// TIA Portal V18 program export: 3 tag tables, 0 data types, 3 data blocks, 3 code blocks (in call order from the OBs), 0 instance data blocks

VAR_GLOBAL   // PLC tag table "Default tag table"
   Motor_Contactor AT %Q0.0 : Bool;
   Clock_Byte AT %MB100 : Byte;
   Clock_10Hz AT %M100.0 : Bool;
   Clock_5Hz AT %M100.1 : Bool;
   "Clock_2.5Hz" AT %M100.2 : Bool;
   Clock_2Hz AT %M100.3 : Bool;
   "Clock_1.25Hz" AT %M100.4 : Bool;
   "Clock_0.625Hz" AT %M100.6 : Bool;
   "Clock_0.5Hz" AT %M100.7 : Bool;
END_VAR

VAR_GLOBAL   // PLC tag table "Encoder_Tags"
   HSC_1_Value AT %ID1000 : DInt;   // Giá trị đếm xung thời kỳ thực từ bộ đếm tốc độ cao HSC1   {ExternalWritable false}
END_VAR

VAR_GLOBAL   // PLC tag table "PLC2_Tags"
   MB_ControlWord AT %MW40 : Word;
   MB_FreqSetpoint AT %MW42 : Int;
   MB_StatusWord AT %MW44 : Word;
   MB_ActualSpeed AT %MW46 : Int;
   MB_Error AT %M50.0 : Bool;
   MB_Busy AT %M50.1 : Bool;
   MB_Done AT %M50.2 : Bool;
   MB_Status AT %MW52 : Word;
   iStep AT %MW60 : Int;
   Freq_Temp AT %MD70 : Real;
   Speed_Actual_Temp AT %MD74 : Real;
   FirstScan AT %M101.0 : Bool;
   Clock_1Hz AT %M100.5 : Bool;
   MBCL_Done AT %M51.0 : Bool;
   MBCL_Error AT %M51.1 : Bool;
   MBCL_Status AT %MW54 : Word;
END_VAR

DATA_BLOCK "DB1_NhanTuPLC1"   // DB1
{ S7_Optimized_Access := 'FALSE' }
VERSION : 0.1
// stored: AutoNumber true, IsOnlyStoredInLoadMemory false, IsWriteProtectedInAS false
   VAR
      Speed_SP_fromPLC1 : Real;
      Control_Byte : Bool;
      Reset_Cmd : Bool;
      DIR_Cmd : Bool;
   END_VAR
BEGIN
END_DATA_BLOCK

DATA_BLOCK "DB2_GuiVePLC1"   // DB2
{ S7_Optimized_Access := 'FALSE' }
VERSION : 0.1
// stored: AutoNumber true, IsOnlyStoredInLoadMemory false, IsWriteProtectedInAS false
   VAR
      Speed_Actual_toSend : Real;
      ATV12_Status_toSend : Word;
   END_VAR
BEGIN
END_DATA_BLOCK

DATA_BLOCK "DB3_Encoder"   // DB5
TITLE = Encoder HSC Data Block
{ S7_Optimized_Access := 'FALSE' }
VERSION : 0.1
// Khối dữ liệu chứa tham số và trạng thái Encoder HSC1
// stored: AutoNumber true, IsOnlyStoredInLoadMemory false, IsWriteProtectedInAS false
   VAR
      Encoder_Count_Current : DInt;
      Encoder_Count_Last : DInt;
      Encoder_Count_Delta : DInt;
      Encoder_Count_Delta_Real : Real;
      Encoder_PPR : Real := 1000.0;
      Encoder_Effective_PPR : Real;
      Encoder_SampleTime_s : Real := 0.1;
      Encoder_RPM : Real;
      Encoder_Hz_Raw : Real;
      Encoder_Hz : Real;
      Encoder_Feedback_Selected : Real;
      Encoder_Use_Feedback : Bool := true;
      Encoder_Fault : Bool;
      Encoder_Use_Fourfold : Bool := true;
      Encoder_Motor_Pole_Pairs : Real := 2.0;
      Encoder_Fallback_Active : Bool;
      Encoder_NoPulse_Count : Real;
      Encoder_NoPulse_Limit : Real := 30.0;
   END_VAR
BEGIN
END_DATA_BLOCK

ORGANIZATION_BLOCK "Main"   // OB1, LAD, ProgramCycle
TITLE = "Main Program Sweep (Cycle)"
{ S7_Optimized_Access := 'TRUE' }
VERSION : 0.1
// stored: AutoNumber true, IsIECCheckEnabled false, SetENOAutomatically false
   VAR_INPUT
      Initial_Call : Bool;   // Initial call of this OB
      Remanence : Bool;   // =True, if remanent data are available
   END_VAR
BEGIN

REGION Network 1: Call FC_PLC2_Logic (Convert + Step Advance)
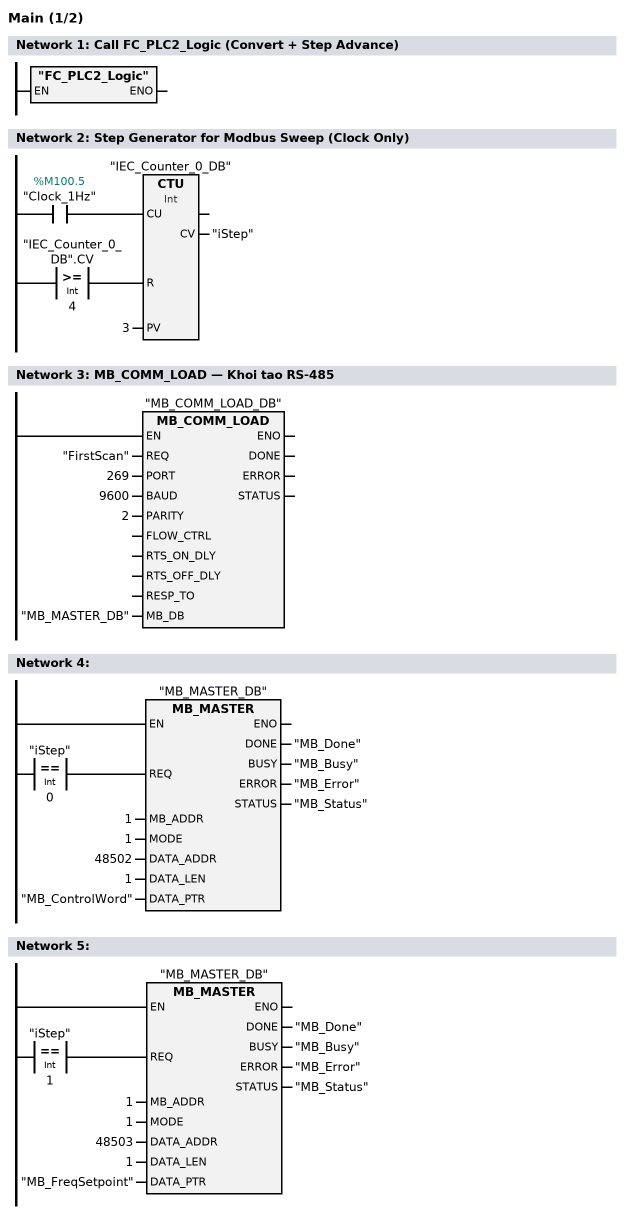
   RUNG wire#powerrail
      "FC_PLC2_Logic"()
   END_RUNG
   // the same network as SCL:
   "FC_PLC2_Logic"();
END_REGION

REGION Network 2: Step Generator for Modbus Sweep (Clock Only)
   RUNG wire#powerrail
      Contact( "Clock_1Hz" )
      { S7_Templates := "value_type := Int" } "IEC_Counter_0_DB".CTU(r := wire#w1, pv := 3, cv => "iStep")
   END_RUNG
   RUNG wire#powerrail
      { S7_Templates := "SrcType := Int" } GE_Contact(in1 := "IEC_Counter_0_DB".CV, in2 := 4)
   END_RUNG wire#w1
   // the same network as SCL:
   "IEC_Counter_0_DB".CTU(CU := "Clock_1Hz", R := "IEC_Counter_0_DB".CV >= 4, PV := 3, CV => "iStep");
END_REGION

REGION Network 3: MB_COMM_LOAD — Khoi tao RS-485
   RUNG wire#powerrail
      "MB_COMM_LOAD_DB".MB_COMM_LOAD(REQ := "FirstScan", PORT := 269, BAUD := 9600, PARITY := 2, FLOW_CTRL :=, RTS_ON_DLY :=, RTS_OFF_DLY :=, RESP_TO :=, MB_DB := "MB_MASTER_DB", DONE =>, ERROR =>, STATUS =>)
   END_RUNG
   // the same network as SCL:
   "MB_COMM_LOAD_DB"(REQ := "FirstScan", PORT := 269, BAUD := 9600, PARITY := 2, MB_DB := "MB_MASTER_DB");   // MB_COMM_LOAD
END_REGION

REGION Network 4
   RUNG wire#powerrail
      "MB_MASTER_DB".MB_MASTER(REQ := wire#w1, MB_ADDR := 1, MODE := 1, DATA_ADDR := 48502, DATA_LEN := 1, DATA_PTR := "MB_ControlWord", DONE => "MB_Done", BUSY => "MB_Busy", ERROR => "MB_Error", STATUS => "MB_Status")
   END_RUNG
   RUNG wire#powerrail
      { S7_Templates := "SrcType := Int" } EQ_Contact(in1 := "iStep", in2 := 0)
   END_RUNG wire#w1
   // the same network as SCL:
   "MB_MASTER_DB"(REQ := "iStep" = 0,   // MB_MASTER
                  MB_ADDR := 1,
                  MODE := 1,
                  DATA_ADDR := 48502,
                  DATA_LEN := 1,
                  DATA_PTR := "MB_ControlWord",
                  DONE => "MB_Done",
                  BUSY => "MB_Busy",
                  ERROR => "MB_Error",
                  STATUS => "MB_Status");
END_REGION

REGION Network 5
   RUNG wire#powerrail
      "MB_MASTER_DB".MB_MASTER(REQ := wire#w1, MB_ADDR := 1, MODE := 1, DATA_ADDR := 48503, DATA_LEN := 1, DATA_PTR := "MB_FreqSetpoint", DONE => "MB_Done", BUSY => "MB_Busy", ERROR => "MB_Error", STATUS => "MB_Status")
   END_RUNG
   RUNG wire#powerrail
      { S7_Templates := "SrcType := Int" } EQ_Contact(in1 := "iStep", in2 := 1)
   END_RUNG wire#w1
   // the same network as SCL:
   "MB_MASTER_DB"(REQ := "iStep" = 1,   // MB_MASTER
                  MB_ADDR := 1,
                  MODE := 1,
                  DATA_ADDR := 48503,
                  DATA_LEN := 1,
                  DATA_PTR := "MB_FreqSetpoint",
                  DONE => "MB_Done",
                  BUSY => "MB_Busy",
                  ERROR => "MB_Error",
                  STATUS => "MB_Status");
END_REGION

REGION Network 6
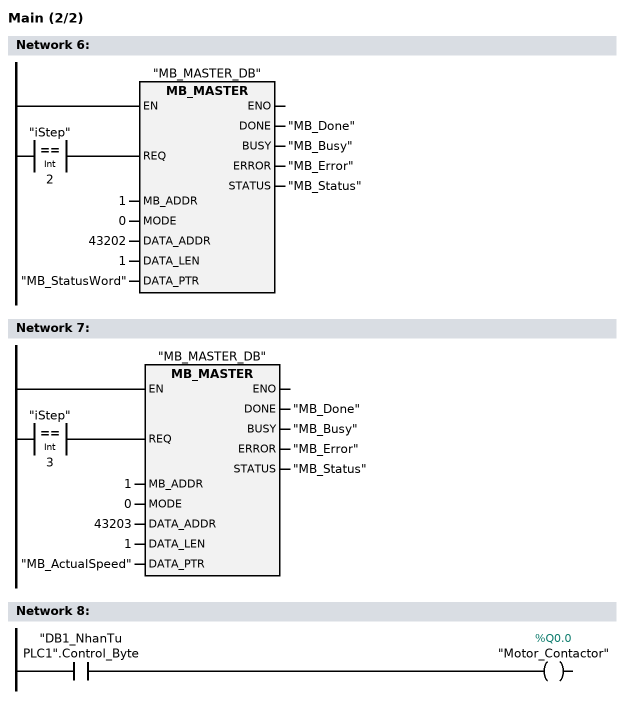
   RUNG wire#powerrail
      "MB_MASTER_DB".MB_MASTER(REQ := wire#w1, MB_ADDR := 1, MODE := 0, DATA_ADDR := 43202, DATA_LEN := 1, DATA_PTR := "MB_StatusWord", DONE => "MB_Done", BUSY => "MB_Busy", ERROR => "MB_Error", STATUS => "MB_Status")
   END_RUNG
   RUNG wire#powerrail
      { S7_Templates := "SrcType := Int" } EQ_Contact(in1 := "iStep", in2 := 2)
   END_RUNG wire#w1
   // the same network as SCL:
   "MB_MASTER_DB"(REQ := "iStep" = 2,   // MB_MASTER
                  MB_ADDR := 1,
                  MODE := 0,
                  DATA_ADDR := 43202,
                  DATA_LEN := 1,
                  DATA_PTR := "MB_StatusWord",
                  DONE => "MB_Done",
                  BUSY => "MB_Busy",
                  ERROR => "MB_Error",
                  STATUS => "MB_Status");
END_REGION

REGION Network 7
   RUNG wire#powerrail
      "MB_MASTER_DB".MB_MASTER(REQ := wire#w1, MB_ADDR := 1, MODE := 0, DATA_ADDR := 43203, DATA_LEN := 1, DATA_PTR := "MB_ActualSpeed", DONE => "MB_Done", BUSY => "MB_Busy", ERROR => "MB_Error", STATUS => "MB_Status")
   END_RUNG
   RUNG wire#powerrail
      { S7_Templates := "SrcType := Int" } EQ_Contact(in1 := "iStep", in2 := 3)
   END_RUNG wire#w1
   // the same network as SCL:
   "MB_MASTER_DB"(REQ := "iStep" = 3,   // MB_MASTER
                  MB_ADDR := 1,
                  MODE := 0,
                  DATA_ADDR := 43203,
                  DATA_LEN := 1,
                  DATA_PTR := "MB_ActualSpeed",
                  DONE => "MB_Done",
                  BUSY => "MB_Busy",
                  ERROR => "MB_Error",
                  STATUS => "MB_Status");
END_REGION

REGION Network 8
   RUNG wire#powerrail
      Contact( "DB1_NhanTuPLC1".Control_Byte )
      Coil( "Motor_Contactor" )
   END_RUNG
   // the same network as SCL:
   "Motor_Contactor" := "DB1_NhanTuPLC1".Control_Byte;
END_REGION
END_ORGANIZATION_BLOCK

FUNCTION "FC_PLC2_Logic" : Void   // FC10, LAD
{ S7_Optimized_Access := 'TRUE' }
VERSION : 0.1
// stored: AutoNumber true, IsIECCheckEnabled false, SetENOAutomatically false, UDAEnableTagReadback false
BEGIN

REGION Network 1: Freq Scale: SP x 10
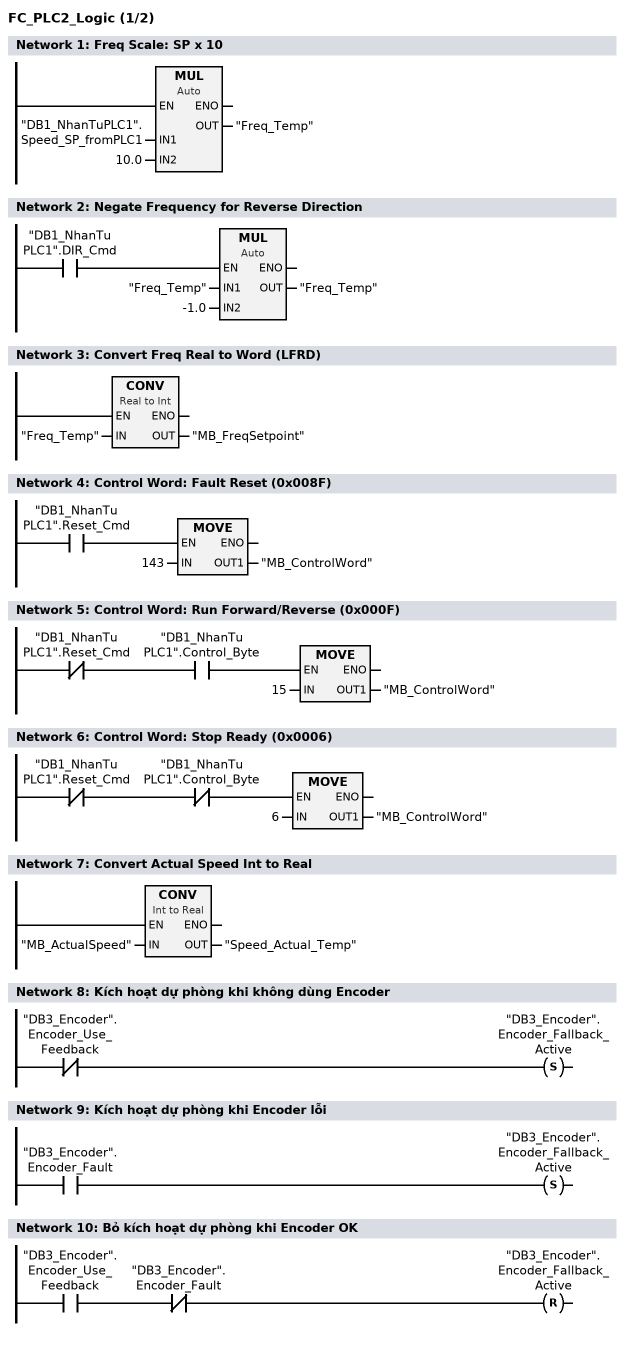
   RUNG wire#powerrail
      { S7_GenerateENO := "TRUE" } Mul(in1 := "DB1_NhanTuPLC1".Speed_SP_fromPLC1, in2 := 10.0, out => "Freq_Temp")
   END_RUNG
   // the same network as SCL:
   "Freq_Temp" := "DB1_NhanTuPLC1".Speed_SP_fromPLC1 * 10.0;
END_REGION

REGION Network 2: Negate Frequency for Reverse Direction
   RUNG wire#powerrail
      Contact( "DB1_NhanTuPLC1".DIR_Cmd )
      { S7_GenerateENO := "TRUE" } Mul(in1 := "Freq_Temp", in2 := -1.0, out => "Freq_Temp")
   END_RUNG
   // the same network as SCL:
   IF "DB1_NhanTuPLC1".DIR_Cmd THEN "Freq_Temp" := "Freq_Temp" * (-1.0); END_IF;
END_REGION

REGION Network 3: Convert Freq Real to Word (LFRD)
   RUNG wire#powerrail
      { S7_Templates := "[SrcType := Real, DestType := Int]"; S7_GenerateENO := "TRUE" } Convert(in := "Freq_Temp", out => "MB_FreqSetpoint")
   END_RUNG
   // the same network as SCL:
   "MB_FreqSetpoint" := REAL_TO_INT("Freq_Temp");
END_REGION

REGION Network 4: Control Word: Fault Reset (0x008F)
   RUNG wire#powerrail
      Contact( "DB1_NhanTuPLC1".Reset_Cmd )
      { S7_GenerateENO := "TRUE" } Move(in := 143, out1 => "MB_ControlWord")
   END_RUNG
   // the same network as SCL:
   IF "DB1_NhanTuPLC1".Reset_Cmd THEN "MB_ControlWord" := 143; END_IF;
END_REGION

REGION Network 5: Control Word: Run Forward/Reverse (0x000F)
   RUNG wire#powerrail
      I_Contact( "DB1_NhanTuPLC1".Reset_Cmd )
      Contact( "DB1_NhanTuPLC1".Control_Byte )
      { S7_GenerateENO := "TRUE" } Move(in := 15, out1 => "MB_ControlWord")
   END_RUNG
   // the same network as SCL:
   IF NOT "DB1_NhanTuPLC1".Reset_Cmd AND "DB1_NhanTuPLC1".Control_Byte THEN "MB_ControlWord" := 15; END_IF;
END_REGION

REGION Network 6: Control Word: Stop Ready (0x0006)
   RUNG wire#powerrail
      I_Contact( "DB1_NhanTuPLC1".Reset_Cmd )
      I_Contact( "DB1_NhanTuPLC1".Control_Byte )
      { S7_GenerateENO := "TRUE" } Move(in := 6, out1 => "MB_ControlWord")
   END_RUNG
   // the same network as SCL:
   IF NOT "DB1_NhanTuPLC1".Reset_Cmd AND NOT "DB1_NhanTuPLC1".Control_Byte THEN
       "MB_ControlWord" := 6;
   END_IF;
END_REGION

REGION Network 7: Convert Actual Speed Int to Real
   RUNG wire#powerrail
      { S7_Templates := "[SrcType := Int, DestType := Real]"; S7_GenerateENO := "TRUE" } Convert(in := "MB_ActualSpeed", out => "Speed_Actual_Temp")
   END_RUNG
   // the same network as SCL:
   "Speed_Actual_Temp" := INT_TO_REAL("MB_ActualSpeed");
END_REGION

REGION Network 8: Kích hoạt dự phòng khi không dùng Encoder
   RUNG wire#powerrail
      I_Contact( "DB3_Encoder".Encoder_Use_Feedback )
      S_Coil( "DB3_Encoder".Encoder_Fallback_Active )
   END_RUNG
   // the same network as SCL:
   IF NOT "DB3_Encoder".Encoder_Use_Feedback THEN "DB3_Encoder".Encoder_Fallback_Active := TRUE; END_IF;
END_REGION

REGION Network 9: Kích hoạt dự phòng khi Encoder lỗi
   RUNG wire#powerrail
      Contact( "DB3_Encoder".Encoder_Fault )
      S_Coil( "DB3_Encoder".Encoder_Fallback_Active )
   END_RUNG
   // the same network as SCL:
   IF "DB3_Encoder".Encoder_Fault THEN "DB3_Encoder".Encoder_Fallback_Active := TRUE; END_IF;
END_REGION

REGION Network 10: Bỏ kích hoạt dự phòng khi Encoder OK
   RUNG wire#powerrail
      Contact( "DB3_Encoder".Encoder_Use_Feedback )
      I_Contact( "DB3_Encoder".Encoder_Fault )
      R_Coil( "DB3_Encoder".Encoder_Fallback_Active )
   END_RUNG
   // the same network as SCL:
   IF "DB3_Encoder".Encoder_Use_Feedback AND NOT "DB3_Encoder".Encoder_Fault THEN
       "DB3_Encoder".Encoder_Fallback_Active := FALSE;
   END_IF;
END_REGION

REGION Network 11: Gửi tốc độ thực về PLC_1 chế độ bình thường
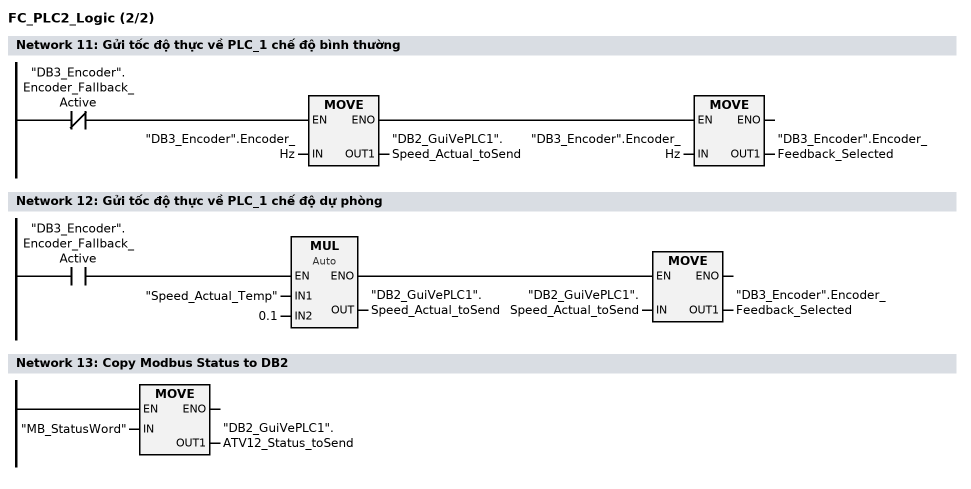
   RUNG wire#powerrail
      I_Contact( "DB3_Encoder".Encoder_Fallback_Active )
      { S7_GenerateENO := "TRUE" } Move(in := "DB3_Encoder".Encoder_Hz, out1 => "DB2_GuiVePLC1".Speed_Actual_toSend)
      { S7_GenerateENO := "TRUE" } Move(in := "DB3_Encoder".Encoder_Hz, out1 => "DB3_Encoder".Encoder_Feedback_Selected)
   END_RUNG
   // the same network as SCL:
   // ENO of a box is taken as its EN; it also drops when the box reports an error
   IF NOT "DB3_Encoder".Encoder_Fallback_Active THEN
       "DB2_GuiVePLC1".Speed_Actual_toSend := "DB3_Encoder".Encoder_Hz;
       "DB3_Encoder".Encoder_Feedback_Selected := "DB3_Encoder".Encoder_Hz;
   END_IF;
END_REGION

REGION Network 12: Gửi tốc độ thực về PLC_1 chế độ dự phòng
   RUNG wire#powerrail
      Contact( "DB3_Encoder".Encoder_Fallback_Active )
      { S7_GenerateENO := "TRUE" } Mul(in1 := "Speed_Actual_Temp", in2 := 0.1, out => "DB2_GuiVePLC1".Speed_Actual_toSend)
      { S7_GenerateENO := "TRUE" } Move(in := "DB2_GuiVePLC1".Speed_Actual_toSend, out1 => "DB3_Encoder".Encoder_Feedback_Selected)
   END_RUNG
   // the same network as SCL:
   // ENO of a box is taken as its EN; it also drops when the box reports an error
   IF "DB3_Encoder".Encoder_Fallback_Active THEN
       "DB2_GuiVePLC1".Speed_Actual_toSend := "Speed_Actual_Temp" * 0.1;
       "DB3_Encoder".Encoder_Feedback_Selected := "DB2_GuiVePLC1".Speed_Actual_toSend;
   END_IF;
END_REGION

REGION Network 13: Copy Modbus Status to DB2
   RUNG wire#powerrail
      { S7_GenerateENO := "TRUE" } Move(in := "MB_StatusWord", out1 => "DB2_GuiVePLC1".ATV12_Status_toSend)
   END_RUNG
   // the same network as SCL:
   "DB2_GuiVePLC1".ATV12_Status_toSend := "MB_StatusWord";
END_REGION
END_FUNCTION

ORGANIZATION_BLOCK "OB30_Encoder_100ms"   // OB30, LAD, CyclicInterrupt
{ S7_Optimized_Access := 'TRUE' }
VERSION : 0.1
// stored: AutoNumber true, IsIECCheckEnabled false, SetENOAutomatically false
   VAR_INPUT
      Initial_Call : Bool;   // Initial call of this OB
      Event_Count : Int;   // Events discarded
   END_VAR
BEGIN

REGION Network 1: Đọc giá trị HSC và tính Delta Count
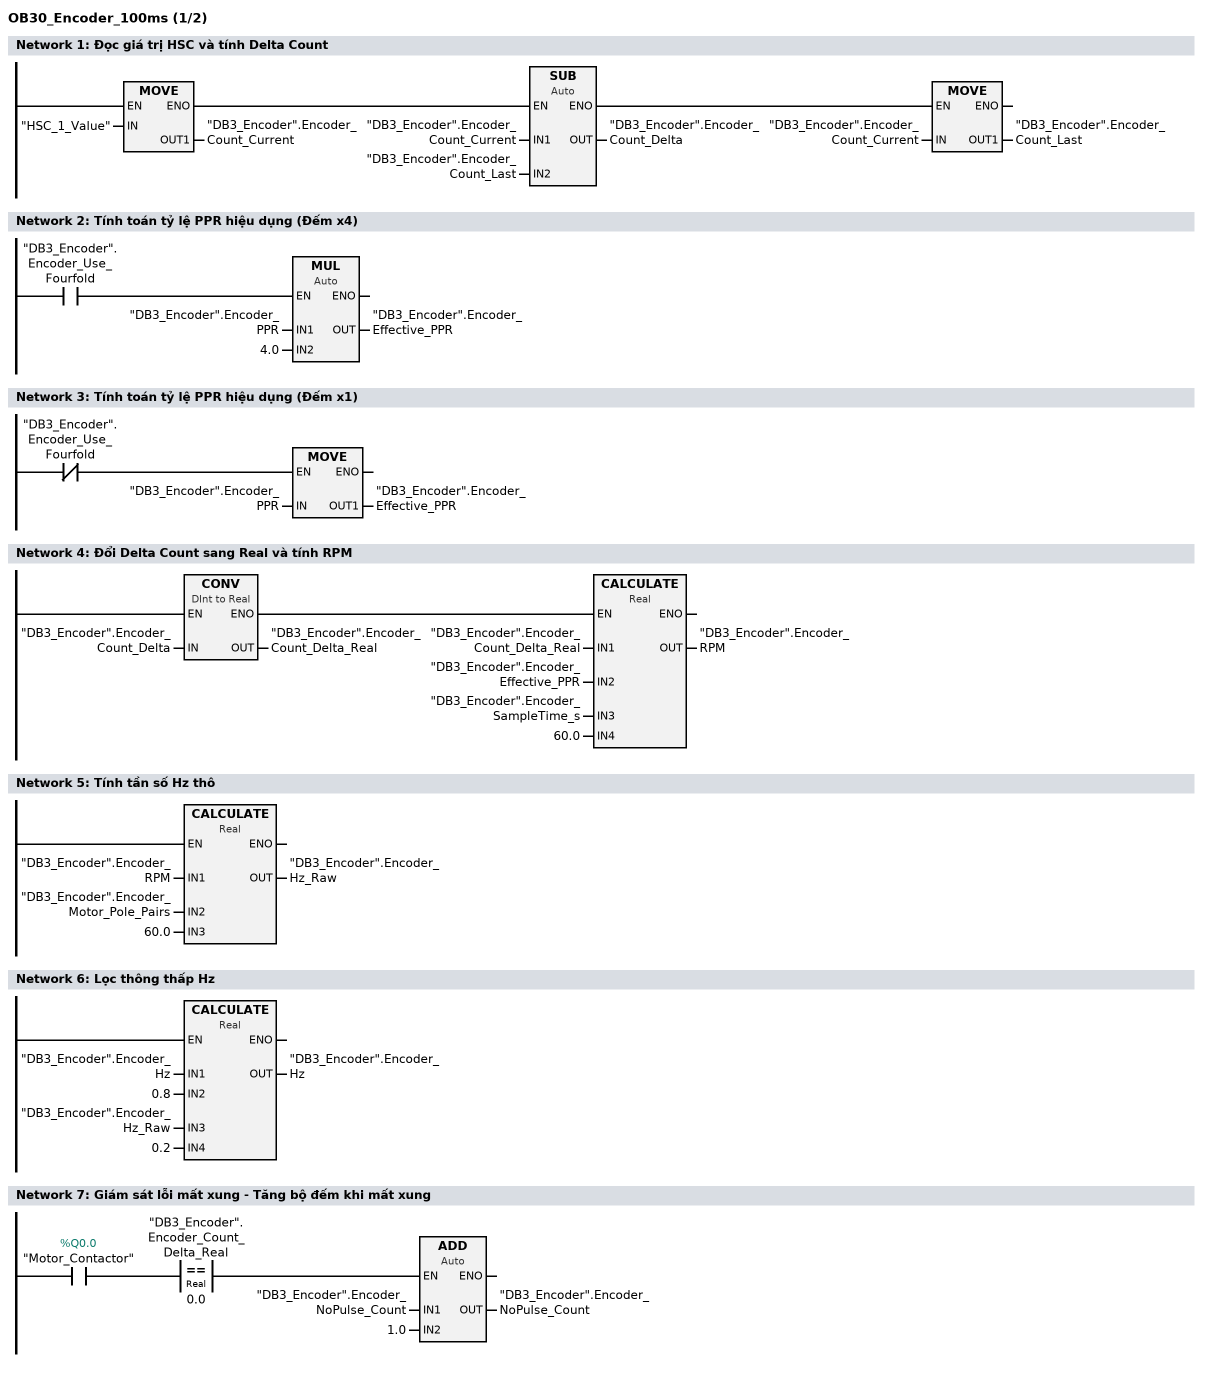
   RUNG wire#powerrail
      { S7_GenerateENO := "TRUE" } Move(in := "HSC_1_Value", out1 => "DB3_Encoder".Encoder_Count_Current)
      { S7_GenerateENO := "TRUE" } Sub(in1 := "DB3_Encoder".Encoder_Count_Current, in2 := "DB3_Encoder".Encoder_Count_Last, out => "DB3_Encoder".Encoder_Count_Delta)
      { S7_GenerateENO := "TRUE" } Move(in := "DB3_Encoder".Encoder_Count_Current, out1 => "DB3_Encoder".Encoder_Count_Last)
   END_RUNG
   // the same network as SCL:
   // ENO of a box is taken as its EN; it also drops when the box reports an error
   "DB3_Encoder".Encoder_Count_Current := "HSC_1_Value";
   "DB3_Encoder".Encoder_Count_Delta := "DB3_Encoder".Encoder_Count_Current - "DB3_Encoder".Encoder_Count_Last;
   "DB3_Encoder".Encoder_Count_Last := "DB3_Encoder".Encoder_Count_Current;
END_REGION

REGION Network 2: Tính toán tỷ lệ PPR hiệu dụng (Đếm x4)
   RUNG wire#powerrail
      Contact( "DB3_Encoder".Encoder_Use_Fourfold )
      { S7_GenerateENO := "TRUE" } Mul(in1 := "DB3_Encoder".Encoder_PPR, in2 := 4.0, out => "DB3_Encoder".Encoder_Effective_PPR)
   END_RUNG
   // the same network as SCL:
   IF "DB3_Encoder".Encoder_Use_Fourfold THEN
       "DB3_Encoder".Encoder_Effective_PPR := "DB3_Encoder".Encoder_PPR * 4.0;
   END_IF;
END_REGION

REGION Network 3: Tính toán tỷ lệ PPR hiệu dụng (Đếm x1)
   RUNG wire#powerrail
      I_Contact( "DB3_Encoder".Encoder_Use_Fourfold )
      { S7_GenerateENO := "TRUE" } Move(in := "DB3_Encoder".Encoder_PPR, out1 => "DB3_Encoder".Encoder_Effective_PPR)
   END_RUNG
   // the same network as SCL:
   IF NOT "DB3_Encoder".Encoder_Use_Fourfold THEN
       "DB3_Encoder".Encoder_Effective_PPR := "DB3_Encoder".Encoder_PPR;
   END_IF;
END_REGION

REGION Network 4: Đổi Delta Count sang Real và tính RPM
   RUNG wire#powerrail
      { S7_Templates := "[SrcType := DInt, DestType := Real]"; S7_GenerateENO := "TRUE" } Convert(in := "DB3_Encoder".Encoder_Count_Delta, out => "DB3_Encoder".Encoder_Count_Delta_Real)
      { S7_Templates := "SrcType := Real"; S7_GenerateENO := "TRUE"; S7_Expression := "(IN1 * IN4) / (IN2 * IN3)" } Calculate(in1 := "DB3_Encoder".Encoder_Count_Delta_Real, in2 := "DB3_Encoder".Encoder_Effective_PPR, in3 := "DB3_Encoder".Encoder_SampleTime_s, in4 := 60.0, out => "DB3_Encoder".Encoder_RPM)
   END_RUNG
   // the same network as SCL:
   // ENO of a box is taken as its EN; it also drops when the box reports an error
   "DB3_Encoder".Encoder_Count_Delta_Real := DINT_TO_REAL("DB3_Encoder".Encoder_Count_Delta);
   "DB3_Encoder".Encoder_RPM := ("DB3_Encoder".Encoder_Count_Delta_Real * 60.0) / ("DB3_Encoder".Encoder_Effective_PPR * "DB3_Encoder".Encoder_SampleTime_s);
END_REGION

REGION Network 5: Tính tần số Hz thô
   RUNG wire#powerrail
      { S7_Templates := "SrcType := Real"; S7_GenerateENO := "TRUE"; S7_Expression := "(IN1 * IN2) / IN3" } Calculate(in1 := "DB3_Encoder".Encoder_RPM, in2 := "DB3_Encoder".Encoder_Motor_Pole_Pairs, in3 := 60.0, out => "DB3_Encoder".Encoder_Hz_Raw)
   END_RUNG
   // the same network as SCL:
   "DB3_Encoder".Encoder_Hz_Raw := ("DB3_Encoder".Encoder_RPM * "DB3_Encoder".Encoder_Motor_Pole_Pairs) / 60.0;
END_REGION

REGION Network 6: Lọc thông thấp Hz
   RUNG wire#powerrail
      { S7_Templates := "SrcType := Real"; S7_GenerateENO := "TRUE"; S7_Expression := "(IN1 * IN2) + (IN3 * IN4)" } Calculate(in1 := "DB3_Encoder".Encoder_Hz, in2 := 0.8, in3 := "DB3_Encoder".Encoder_Hz_Raw, in4 := 0.2, out => "DB3_Encoder".Encoder_Hz)
   END_RUNG
   // the same network as SCL:
   "DB3_Encoder".Encoder_Hz := ("DB3_Encoder".Encoder_Hz * 0.8) + ("DB3_Encoder".Encoder_Hz_Raw * 0.2);
END_REGION

REGION Network 7: Giám sát lỗi mất xung - Tăng bộ đếm khi mất xung
   RUNG wire#powerrail
      Contact( "Motor_Contactor" )
      { S7_Templates := "SrcType := Real" } EQ_Contact(in1 := "DB3_Encoder".Encoder_Count_Delta_Real, in2 := 0.0)
      { S7_GenerateENO := "TRUE" } Add(in1 := "DB3_Encoder".Encoder_NoPulse_Count, in2 := 1.0, out => "DB3_Encoder".Encoder_NoPulse_Count)
   END_RUNG
   // the same network as SCL:
   IF "Motor_Contactor" AND ("DB3_Encoder".Encoder_Count_Delta_Real = 0.0) THEN
       "DB3_Encoder".Encoder_NoPulse_Count := "DB3_Encoder".Encoder_NoPulse_Count + 1.0;
   END_IF;
END_REGION

REGION Network 8: Giám sát lỗi mất xung - Reset bộ đếm khi có xung
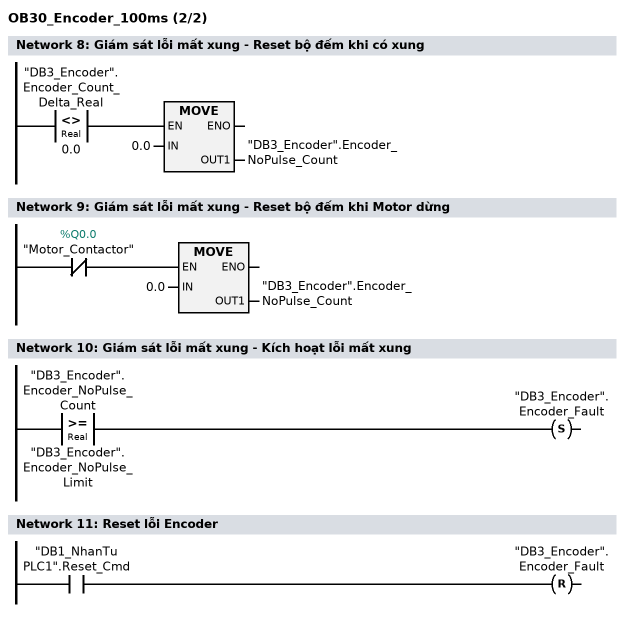
   RUNG wire#powerrail
      { S7_Templates := "SrcType := Real" } NE_Contact(in1 := "DB3_Encoder".Encoder_Count_Delta_Real, in2 := 0.0)
      { S7_GenerateENO := "TRUE" } Move(in := 0.0, out1 => "DB3_Encoder".Encoder_NoPulse_Count)
   END_RUNG
   // the same network as SCL:
   IF "DB3_Encoder".Encoder_Count_Delta_Real <> 0.0 THEN "DB3_Encoder".Encoder_NoPulse_Count := 0.0; END_IF;
END_REGION

REGION Network 9: Giám sát lỗi mất xung - Reset bộ đếm khi Motor dừng
   RUNG wire#powerrail
      I_Contact( "Motor_Contactor" )
      { S7_GenerateENO := "TRUE" } Move(in := 0.0, out1 => "DB3_Encoder".Encoder_NoPulse_Count)
   END_RUNG
   // the same network as SCL:
   IF NOT "Motor_Contactor" THEN "DB3_Encoder".Encoder_NoPulse_Count := 0.0; END_IF;
END_REGION

REGION Network 10: Giám sát lỗi mất xung - Kích hoạt lỗi mất xung
   RUNG wire#powerrail
      { S7_Templates := "SrcType := Real" } GE_Contact(in1 := "DB3_Encoder".Encoder_NoPulse_Count, in2 := "DB3_Encoder".Encoder_NoPulse_Limit)
      S_Coil( "DB3_Encoder".Encoder_Fault )
   END_RUNG
   // the same network as SCL:
   IF "DB3_Encoder".Encoder_NoPulse_Count >= "DB3_Encoder".Encoder_NoPulse_Limit THEN
       "DB3_Encoder".Encoder_Fault := TRUE;
   END_IF;
END_REGION

REGION Network 11: Reset lỗi Encoder
   RUNG wire#powerrail
      Contact( "DB1_NhanTuPLC1".Reset_Cmd )
      R_Coil( "DB3_Encoder".Encoder_Fault )
   END_RUNG
   // the same network as SCL:
   IF "DB1_NhanTuPLC1".Reset_Cmd THEN "DB3_Encoder".Encoder_Fault := FALSE; END_IF;
END_REGION
END_ORGANIZATION_BLOCK
